Fanuc KAREL source: RNUMREG_SEND.kl

PROGRAM T
%NOLOCKGROUP
VAR
 v0 : STRING[40]
 v1 : INTEGER
 v2 : INTEGER
 v3 : INTEGER
 v4 : INTEGER
BEGIN
 RNUMREG_SEND(v0, v1, v2, v3, v4)
END T
